# EPICS autosave request: galilDmc30017App/Db/galil_dmc30017_digital_in_0_3.req
# The files listed here are located at <GALIL support top>/GalilSup/Db
# as they are provided by the Galil Support Module

# Digital input bits 0-3
file "galil_digital_in_bit.req" P=$(P), R=$(DIG_IN0)
file "galil_digital_in_bit.req" P=$(P), R=$(DIG_IN1)
file "galil_digital_in_bit.req" P=$(P), R=$(DIG_IN2)
file "galil_digital_in_bit.req" P=$(P), R=$(DIG_IN3)
